{attribute addProperty BoxType "EL3312-0000-0018"}
{attribute addProperty Id "TC_Inputs_ChannelAT %I*ARRAY[0..1] OF TC_Inputs_Channel_FFD159D66480WcStateAT %I*WcState_F855686C1620InfoDataAT %I*InfoData_BC63D37F80100"}
{attribute addProperty CRC "1460358681"}
{attribute addProperty SizeInBites "160"}
{attribute addProperty SizeInBytes "20"}
TYPE EL3312_322B5855 :
STRUCT
	{attribute addProperty Name "TC_Inputs_Channel"}
	TC_Inputs_Channel : ARRAY[0..1] OF TC_Inputs_Channel_FFD159D6;
	{attribute addProperty Name "WcState"}
	WcState : WcState_F855686C;
	{attribute addProperty Name "InfoData"}
	InfoData : InfoData_BC63D37F;
END_STRUCT
END_TYPE

(* stored: Version 1.2.0.0, ProductVersion 3.1.4024.9
   DUT EL3312_322B5855: Id {4eeb70c4-4787-4fd2-b3ba-e3052dc1229b} *)
